FUNCTION_BLOCK FB_SecondaryControlStartPos
VAR_INPUT
	bEnable 						: BOOL; 
	fPosition						: LREAL;
	fStartPosition					: LREAL;
	
	eStatus 						: BOOL; //E_Status;
END_VAR
VAR_OUTPUT
	bStartPosOK						: BOOL;
	fDisplacementControlSignal		: LREAL;
	bOpenBreak						: BOOL;
END_VAR
VAR PERSISTENT
	fProportionalGain 				: LREAL;
	fIntegralGain					: LREAL;
	fDerivateGain					: LREAL;
END_VAR
VAR
	fbPID_controller				: FB_PID_controller;
	fPosition_error					: LREAL;
	fProportinalGain_output			: LREAL;
	fIntegralGain_output			: LREAL;
	fDerivateGain_output			: LREAL;
    bEnableValveOutputDisp			: BOOL;	
END_VAR

IF eStatus AND G_Engineer_HMI.bSecondaryStartPosEnable THEN
	bOpenBreak	:= TRUE;
ELSE
	bOpenBreak := FALSE;
END_IF

IF bEnable THEN 
	
fPosition_error := fStartPosition - fPosition;

G_Motion_Control.fPosition_error_StartDisplacement := fPosition_error; 

// Write to HMI
//PGain:
IF NOT(G_Engineer_HMI.bPenable_dis_write) THEN
	G_Engineer_HMI.fProportionalgain_dis := fProportionalGain; // SKjønner ikke helt det her
ELSE
	fProportionalGain := G_Engineer_HMI.fProportionalgain_dis;
END_IF

//IGain: 
IF NOT(G_Engineer_HMI.bIenable_dis_write) THEN
	G_Engineer_HMI.fIntegralgain_dis := fIntegralGain;
ELSE
	fIntegralGain := G_Engineer_HMI.fIntegralgain_dis;
END_IF

fbPID_controller(
		ssMethodType := BOOL_TO_SINT(bEnable),
		error := fPosition_error,
		Int_error_threshold := G_PID_Tuning.Int_error_threshold,
		P_enable := G_Engineer_HMI.bPenable_dis,
		I_enable := G_Engineer_HMI.bIenable_dis,
		D_enable := FALSE,
		K_p := fProportionalGain,
		K_i := fIntegralGain,
		K_d := fDerivateGain,
		P_output => fProportinalGain_output,
		I_output => fIntegralGain_output,
		D_output => fDerivateGain_output
		);
		
			//Error times PGain
	fProportinalGain_output := fProportinalGain_output;
	G_PID_Tuning.fProportinalGain_output_dis := fProportinalGain_output;
	//Error times IGain
	fIntegralGain_output := fIntegralGain_output;
	G_PID_Tuning.fIntegralGain_output_dis := fIntegralGain_output;
	//Error times DGain
	fDerivateGain_output := fDerivateGain_output;
	G_PID_Tuning.fDerivateGain_output_dis := fDerivateGain_output;
	
	//Normalized Outputsignal
		
	fDisplacementControlSignal := LIMIT(-1, 1*(fProportinalGain_output + fIntegralGain_output + fDerivateGain_output), 1);
	G_PID_Tuning.PID_output_dis := fDisplacementControlSignal	;			
	
	IF ABS(fPosition_error) < 0.05 THEN
		bStartPosOK := TRUE;
	END_IF
		
ELSE
	bStartPosOK := FALSE;

END_IF

END_FUNCTION_BLOCK

(* stored: Version 1.1.0.1
   POU FB_SecondaryControlStartPos: Id {8eba5c06-ee19-44b5-b58c-05e2066444b9}, SpecialFunc None *)
